{region '#Template'}
	{attribute 'Category' := 'Universal'}
	{attribute 'Version' := '0.0.1.0'}
	{attribute 'Tags' := 'Universal, Control, Anti-blocking protection'}
	{attribute 'Description' := 'Antiblockierschutz 	// Anti-blocking protection'}
{endregion}
FUNCTION_BLOCK FB_BA_AntiBlocking EXTENDS FB_BA_View
VAR_INPUT
	bFdb					: BOOL;	
	bExtReq					: BOOL;
	bLock					: BOOL;
END_VAR
VAR_OUTPUT
	bQ						: BOOL;
END_VAR
VAR_INPUT CONSTANT PERSISTENT
	{attribute 'parameterCategory' := 'Operation'}
	bEn : BOOL := TRUE;
END_VAR
VAR_INPUT CONSTANT
	IdlePrd					: FB_BA_AV_Op;									 
	ImpulseLength			: FB_BA_AV_Op;
END_VAR	
VAR		
	AblkFnct				: FB_BA_AntBlkg;
END_VAR

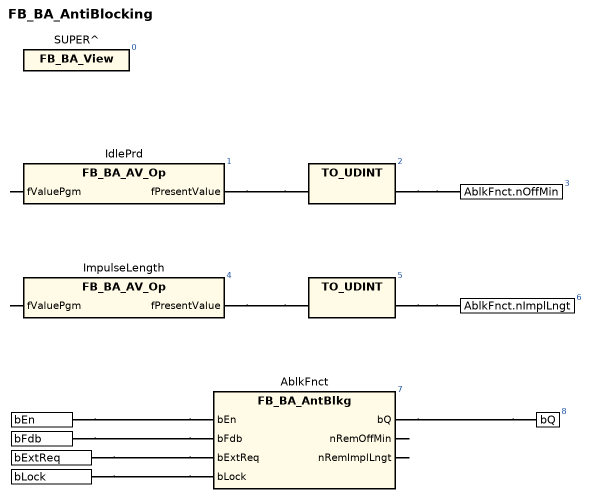
SUPER^(); // FB_BA_View
IdlePrd(); // FB_BA_AV_Op
AblkFnct.nOffMin := TO_UDINT(IdlePrd.fPresentValue);
ImpulseLength(); // FB_BA_AV_Op
AblkFnct.nImplLngt := TO_UDINT(ImpulseLength.fPresentValue);
AblkFnct(bEn := bEn, bFdb := bFdb, bExtReq := bExtReq, bLock := bLock); // FB_BA_AntBlkg
bQ := AblkFnct.bQ;

METHOD FB_init : BOOL
VAR_INPUT
	bInitRetains : BOOL; // if TRUE, the retain variables are initialized (warm start / cold start)
	bInCopyCode : BOOL;  // if TRUE, the instance afterwards gets moved into the copy code (online change)
END_VAR
IdlePrd.iParent					:= THIS^;
IdlePrd.iLabel					:= LblUniControl.AntiBlocking_IdlePeriod;	
IdlePrd.sObjectName				:= '{Idx=01}';								 	 
IdlePrd.eUnit 					:= E_BA_Unit.eTime_Seconds;								 
IdlePrd.fValueRm				:= 604800;
IdlePrd.fCOVIncrement			:= BA2_Param.fDefCOVIncrement;
														 
ImpulseLength.iParent			:= THIS^;
ImpulseLength.iLabel			:= LblUniControl.AntiBlocking_ImpulsLength;	
ImpulseLength.sObjectName		:= '{Idx=01}';								 	 
ImpulseLength.eUnit 			:= E_BA_Unit.eTime_Seconds;								 
ImpulseLength.fValueRm			:= 168;					
ImpulseLength.fCOVIncrement		:= BA2_Param.fDefCOVIncrement;
END_METHOD

END_FUNCTION_BLOCK

(* stored: Version 1.1.0.1, ProductVersion 3.1.4024.6
   POU FB_BA_AntiBlocking: Id {0482996f-e0ae-4d2f-bb97-1f2484f47a56}, SpecialFunc None
   Method FB_init: Id {3ede641e-b421-439b-bed6-180d705bf52d} *)
